{attribute 'GeneratedUsingTerminal: EL2014-0000-0016'}
{attribute addProperty BoxType "EL2014-0000-0016"}
{attribute addProperty Id "EtcSlaveTerminalBaseDIG_Diag_InputsAT %I*DIG_Diag_Inputs_58F3E2A816DIG_Inputs_DeviceAT %I*DIG_Inputs_Device_A1F150A94DIG_OutputsAT %Q*DIG_Outputs_F9744C664WcStateAT %I*WcState_9091E0EB2InfoDataAT %I*InfoData_32EB74EA10"}
{attribute addProperty CRC "2979553674"}
{attribute addProperty Size "36"}
TYPE EL2014_B198618A EXTENDS EtcSlaveTerminalBase :
STRUCT
	{attribute addProperty Name "DIG_Diag_Inputs"}
	DIG_Diag_Inputs : DIG_Diag_Inputs_58F3E2A8;
	{attribute addProperty Name "DIG_Inputs_Device"}
	DIG_Inputs_Device : DIG_Inputs_Device_A1F150A9;
	{attribute addProperty Name "DIG_Outputs"}
	DIG_Outputs : DIG_Outputs_F9744C66;
	{attribute addProperty Name "WcState"}
	WcState : WcState_9091E0EB;
	{attribute addProperty Name "InfoData"}
	InfoData : InfoData_32EB74EA;
END_STRUCT
END_TYPE

(* stored: Version 1.2.0.0, ProductVersion 3.1.4024.9
   DUT EL2014_B198618A: Id {5db7ab93-d19a-4519-ace1-70eb43aff96c} *)
